// LS Electric XG5000 project: 숫자만큼 돌리기
// PLC NewPLC
// module base 0 slot 0: 입출력 모듈:XBC-DR32H (DC 24V 입력, 릴레이 출력 32점)
// module base 0 slot 1: 위치결정 모듈:XBF-PD02A (위치결정 펄스(LD)출력형, 2축)
// module base 0 slot 2: 출력 모듈:XBE-TN/TP16A (트랜지스터 출력, 16점 (싱크출력/소스출력))

PROGRAM NewProgram (task: 스캔 프로그램)

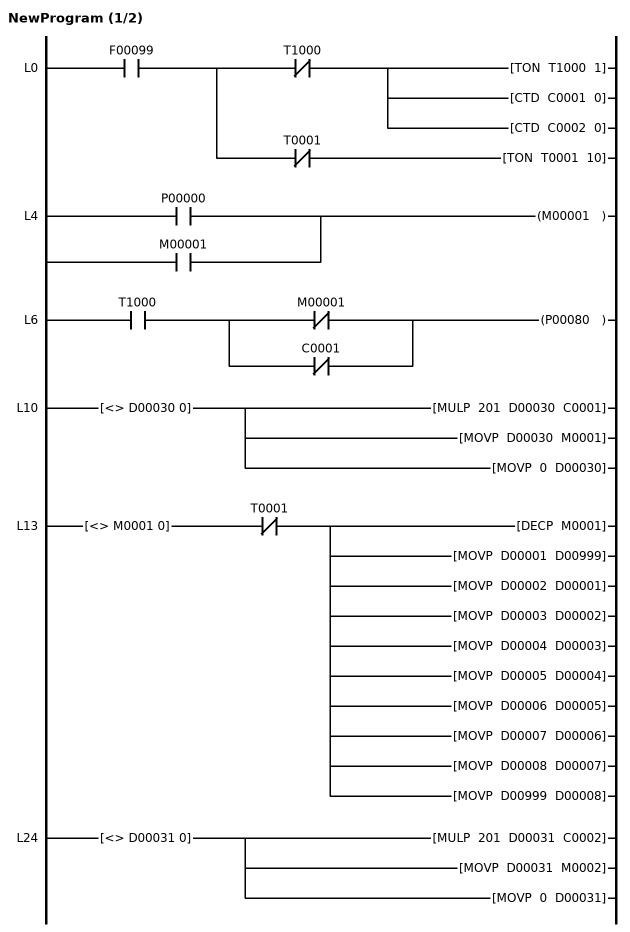
; L0
LOAD      F00099
MPUSH
AND NOT   T1000
TON       T1000 1
CTD       C0001 0
CTD       C0002 0
MPOP
AND NOT   T0001
TON       T0001 10
; L4
LOAD      P00000
OR        M00001
OUT       M00001
; L6
LOAD      T1000
LOAD NOT  M00001
OR NOT    C0001
AND LOAD
OUT       P00080
; L10
LOAD<>    D00030 0
MULP      201 D00030 C0001
MOVP      D00030 M0001
MOVP      0 D00030
; L13
LOAD<>    M0001 0
AND NOT   T0001
DECP      M0001
MOVP      D00001 D00999
MOVP      D00002 D00001
MOVP      D00003 D00002
MOVP      D00004 D00003
MOVP      D00005 D00004
MOVP      D00006 D00005
MOVP      D00007 D00006
MOVP      D00008 D00007
MOVP      D00999 D00008
; L24
LOAD<>    D00031 0
MULP      201 D00031 C0002
MOVP      D00031 M0002
MOVP      0 D00031

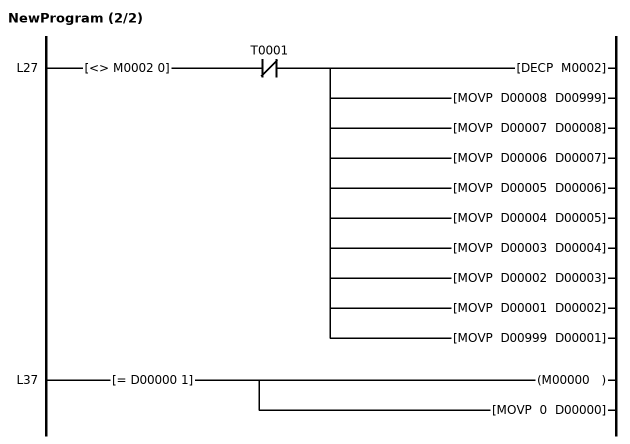
; L27
LOAD<>    M0002 0
AND NOT   T0001
DECP      M0002
MOVP      D00008 D00999
MOVP      D00007 D00008
MOVP      D00006 D00007
MOVP      D00005 D00006
MOVP      D00004 D00005
MOVP      D00003 D00004
MOVP      D00002 D00003
MOVP      D00001 D00002
MOVP      D00999 D00001
; L37
LOAD=     D00000 1
OUT       M00000
MOVP      0 D00000